PROGRAM pouS4Prompts
VAR
	


idbMsgPrompt: FB_CheckMessageBounds;
END_VAR

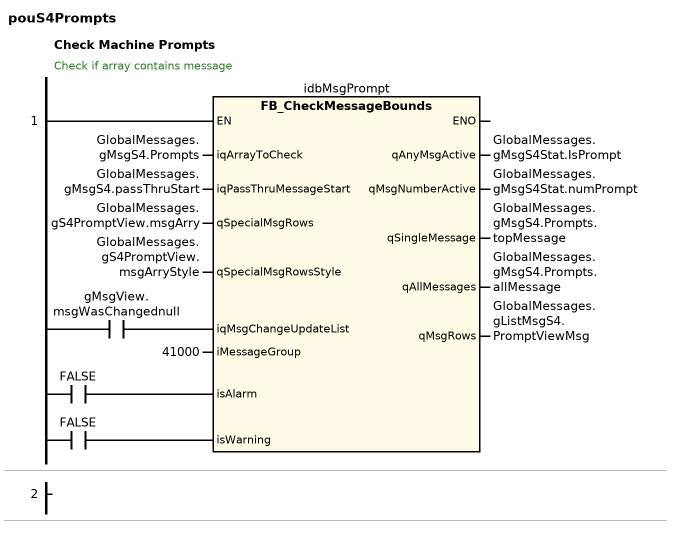
// NETWORK 1: Check Machine Prompts
// Check if array contains message
idbMsgPrompt(
    iqArrayToCheck := GlobalMessages.gMsgS4.Prompts,
    iqPassThruMessageStart := GlobalMessages.gMsgS4.passThruStart,
    qSpecialMsgRows := GlobalMessages.gS4PromptView.msgArry,
    qSpecialMsgRowsStyle := GlobalMessages.gS4PromptView.msgArryStyle,
    iqMsgChangeUpdateList := gMsgView.msgWasChangednull,
    iMessageGroup := 41000,
    isAlarm := FALSE,
    isWarning := FALSE,
    qAnyMsgActive => GlobalMessages.gMsgS4Stat.IsPrompt,
    qMsgNumberActive => GlobalMessages.gMsgS4Stat.numPrompt,
    qSingleMessage => GlobalMessages.gMsgS4.Prompts.topMessage,
    qAllMessages => GlobalMessages.gMsgS4.Prompts.allMessage,
    qMsgRows => GlobalMessages.gListMsgS4.PromptViewMsg); // FB_CheckMessageBounds

// NETWORK 2

END_PROGRAM

(* stored: Version 1.1.0.1, ProductVersion 3.1.4024.11
   POU pouS4Prompts: Id {da1db99f-f4b4-4307-97f8-6ec0cc41de57}, SpecialFunc None *)
